PROGRAM MAIN
VAR
END_VAR

END_PROGRAM

(* stored: Version 1.1.0.1
   POU MAIN: Id {7802ecd8-5171-42d6-a8c4-2a1758873295} *)
